FUNCTION_BLOCK FB_BtnHmiAutoResetType
VAR_INPUT
	xEtat: BOOL;
END_VAR
VAR_OUTPUT
	xRisingEdge: BOOL;
END_VAR
VAR
	fbRTrig: R_Trig;
END_VAR

fbRTrig(CLK:=xEtat);
xRisingEdge:=fbRTrig.Q;
xEtat:=FALSE;

END_FUNCTION_BLOCK

(* stored: Version 1.1.0.1, ProductVersion 3.1.4020.12
   POU FB_BtnHmiAutoResetType: Id {6df7e4dc-4b74-467d-a6b2-5f9d45ed3965}, SpecialFunc None *)
